// TIA Portal project "motor_uygulamasi" (V18)

(* hardware
DEVICE "S7-1200 station_1"  S7-1200 Station
   slot 0: "Rack_0"  S7-1200 Rack  Rack  V1.0
   slot 1: "PLC_1"  CPU 1214C AC/DC/Rly  6ES7 214-1BG40-0XB0  V4.6
*)

// ===== PLC "PLC_1"  CPU 1214C AC/DC/Rly =====

VAR_GLOBAL   // PLC tag table "Default tag table"
   "STOP" AT %I0.0 : Bool;
   "START" AT %I0.1 : Bool;
   "YR1" AT %M0.0 : Bool;
   "MOTOR1" AT %Q0.1 : Bool;
   "YR2" AT %M0.1 : Bool;
   "MOTOR2" AT %Q0.2 : Bool;
END_VAR

ORGANIZATION_BLOCK "Main"   // OB1, LAD, ProgramCycle
TITLE = "Main Program Sweep (Cycle)"
{ S7_Optimized_Access := 'TRUE' }
VERSION : 0.1
// UYGULAMA-1: Bir sistemde, 2 adet motor çalistinlacaktir. Start butonuna ilk defa basildiginda sadece 1 nolu motor devreye
// girecek ve strekli çalisacaktir. I. motor çalismaya basladiktan sonra ayni start butonuna ikinci defa basildiginda 2 nolu motor
// devreye girecek ve sürekli çalisacaktir. Stop butonuna basildiginda çalisan motorlar duracaktir.
   VAR_INPUT
      Initial_Call : Bool;   // Initial call of this OB
      Remanence : Bool;   // =True, if remanent data are available
   END_VAR
   VAR_TEMP   // added for the SCL form of the ladder/FBD networks
      _w1 : Bool;
   END_VAR
BEGIN

REGION Network 1
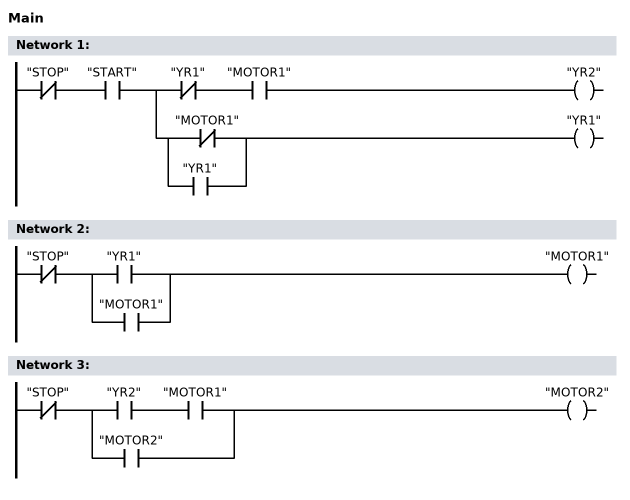
   RUNG wire#powerrail
      I_Contact( "STOP" )
      Contact( "START" )
      wire#w1
      I_Contact( "YR1" )
      Contact( "MOTOR1" )
      Coil( "YR2" )
   END_RUNG
   RUNG wire#w1
      I_Contact( "MOTOR1" )
      wire#w2
      Coil( "YR1" )
   END_RUNG
   RUNG wire#w1
      Contact( "YR1" )
   END_RUNG wire#w2
   // the same network as SCL:
   #_w1 := NOT "STOP" AND "START";
   "YR2" := #_w1 AND NOT "YR1" AND "MOTOR1";
   "YR1" := #_w1 AND (NOT "MOTOR1" OR "YR1");
END_REGION

REGION Network 2
   RUNG wire#powerrail
      I_Contact( "STOP" )
      wire#w1
      Contact( "YR1" )
      wire#w2
      Coil( "MOTOR1" )
   END_RUNG
   RUNG wire#w1
      Contact( "MOTOR1" )
   END_RUNG wire#w2
   // the same network as SCL:
   "MOTOR1" := NOT "STOP" AND ("YR1" OR "MOTOR1");
END_REGION

REGION Network 3
   RUNG wire#powerrail
      I_Contact( "STOP" )
      wire#w1
      Contact( "YR2" )
      Contact( "MOTOR1" )
      wire#w2
      Coil( "MOTOR2" )
   END_RUNG
   RUNG wire#w1
      Contact( "MOTOR2" )
   END_RUNG wire#w2
   // the same network as SCL:
   "MOTOR2" := NOT "STOP" AND (("YR2" AND "MOTOR1") OR "MOTOR2");
END_REGION
END_ORGANIZATION_BLOCK